FUNCTION MS_TO_KMH : REAL
VAR_INPUT
	ms : REAL;
END_VAR


(*
version 1.0	4 Feb 2007
programmer 	hugo
tested by		tobias

this function converts velocities from Meters / Second to Kilometers / hour.

*)

MS_TO_KMH := ms * 3.6;

END_FUNCTION

(* stored: Version 1.1.0.1, ProductVersion 3.1.4024.9
   POU MS_TO_KMH: Id {70dc2ce7-c2da-45d6-b0c5-f7f9d39dfb15}, SpecialFunc None *)
